// LS Electric XG5000 project: 4층_GEMINI
// PLC LSPLC
// module base 0 slot 0: 입출력 모듈:XBC-DR32H (DC 24V 입력, 릴레이 출력 32점)

PROGRAM 6 (task: 스캔 프로그램)

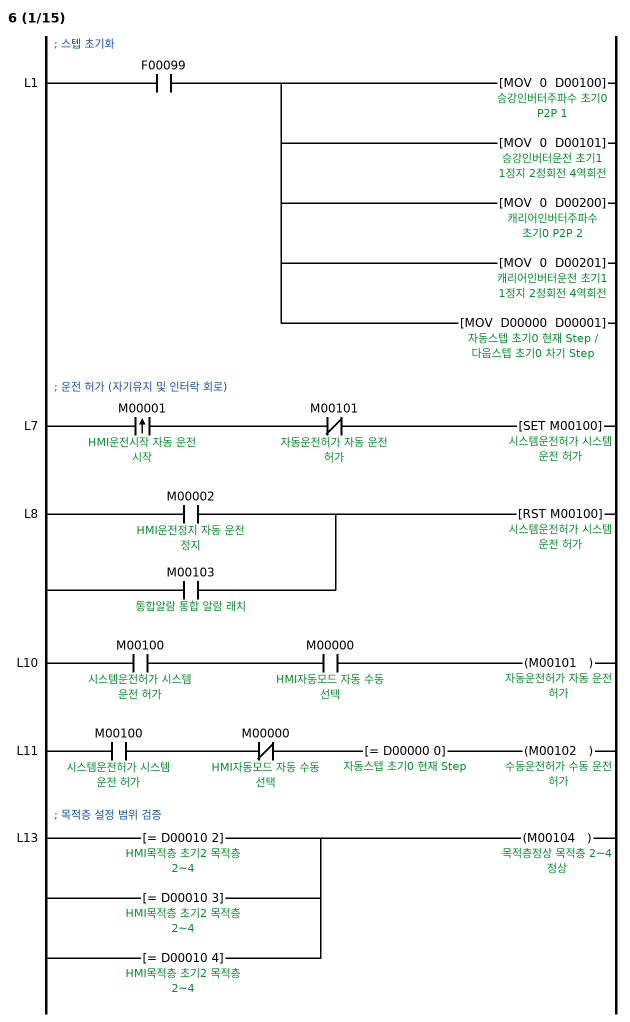
// 스텝 초기화
; L1
LOAD      F00099
MOV       0 D00100	// 승강인버터주파수 초기0 P2P 1
MOV       0 D00101	// 승강인버터운전 초기1 1정지 2정회전 4역회전
MOV       0 D00200	// 캐리어인버터주파수 초기0 P2P 2
MOV       0 D00201	// 캐리어인버터운전 초기1 1정지 2정회전 4역회전
MOV       D00000 D00001	// 자동스텝 초기0 현재 Step / 다음스텝 초기0 차기 Step
// 운전 허가 (자기유지 및 인터락 회로)
; L7
LOADP     M00001	// HMI운전시작 자동 운전 시작
AND NOT   M00101	// 자동운전허가 자동 운전 허가
SET       M00100	// 시스템운전허가 시스템 운전 허가
; L8
LOAD      M00002	// HMI운전정지 자동 운전 정지
OR        M00103	// 통합알람 통합 알람 래치
RST       M00100	// 시스템운전허가 시스템 운전 허가
; L10
LOAD      M00100	// 시스템운전허가 시스템 운전 허가
AND       M00000	// HMI자동모드 자동 수동 선택
OUT       M00101	// 자동운전허가 자동 운전 허가
; L11
LOAD      M00100	// 시스템운전허가 시스템 운전 허가
AND NOT   M00000	// HMI자동모드 자동 수동 선택
AND=      D00000 0	// 자동스텝 초기0 현재 Step
OUT       M00102	// 수동운전허가 수동 운전 허가
// 목적층 설정 범위 검증
; L13
LOAD=     D00010 2	// HMI목적층 초기2 목적층 2~4
OR=       D00010 3	// HMI목적층 초기2 목적층 2~4
OR=       D00010 4	// HMI목적층 초기2 목적층 2~4
OUT       M00104	// 목적층정상 목적층 2~4 정상

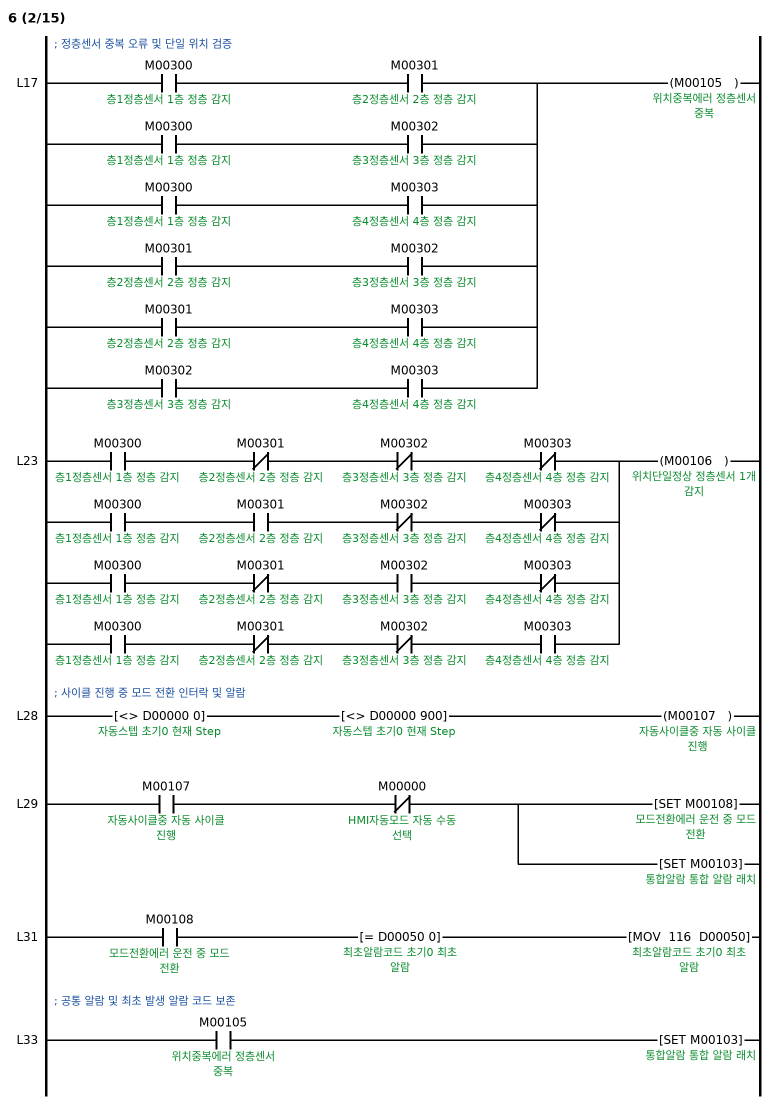
// 정층센서 중복 오류 및 단일 위치 검증
; L17
LOAD      M00300	// 층1정층센서 1층 정층 감지
AND       M00301	// 층2정층센서 2층 정층 감지
LOAD      M00300	// 층1정층센서 1층 정층 감지
AND       M00302	// 층3정층센서 3층 정층 감지
OR LOAD
LOAD      M00300	// 층1정층센서 1층 정층 감지
AND       M00303	// 층4정층센서 4층 정층 감지
OR LOAD
LOAD      M00301	// 층2정층센서 2층 정층 감지
AND       M00302	// 층3정층센서 3층 정층 감지
OR LOAD
LOAD      M00301	// 층2정층센서 2층 정층 감지
AND       M00303	// 층4정층센서 4층 정층 감지
OR LOAD
LOAD      M00302	// 층3정층센서 3층 정층 감지
AND       M00303	// 층4정층센서 4층 정층 감지
OR LOAD
OUT       M00105	// 위치중복에러 정층센서 중복
; L23
LOAD      M00300	// 층1정층센서 1층 정층 감지
AND NOT   M00301	// 층2정층센서 2층 정층 감지
AND NOT   M00302	// 층3정층센서 3층 정층 감지
AND NOT   M00303	// 층4정층센서 4층 정층 감지
LOAD      M00300	// 층1정층센서 1층 정층 감지
AND       M00301	// 층2정층센서 2층 정층 감지
AND NOT   M00302	// 층3정층센서 3층 정층 감지
AND NOT   M00303	// 층4정층센서 4층 정층 감지
OR LOAD
LOAD      M00300	// 층1정층센서 1층 정층 감지
AND NOT   M00301	// 층2정층센서 2층 정층 감지
AND       M00302	// 층3정층센서 3층 정층 감지
AND NOT   M00303	// 층4정층센서 4층 정층 감지
OR LOAD
LOAD      M00300	// 층1정층센서 1층 정층 감지
AND NOT   M00301	// 층2정층센서 2층 정층 감지
AND NOT   M00302	// 층3정층센서 3층 정층 감지
AND       M00303	// 층4정층센서 4층 정층 감지
OR LOAD
OUT       M00106	// 위치단일정상 정층센서 1개 감지
// 사이클 진행 중 모드 전환 인터락 및 알람
; L28
LOAD<>    D00000 0	// 자동스텝 초기0 현재 Step
AND<>     D00000 900	// 자동스텝 초기0 현재 Step
OUT       M00107	// 자동사이클중 자동 사이클 진행
; L29
LOAD      M00107	// 자동사이클중 자동 사이클 진행
AND NOT   M00000	// HMI자동모드 자동 수동 선택
SET       M00108	// 모드전환에러 운전 중 모드 전환
SET       M00103	// 통합알람 통합 알람 래치
; L31
LOAD      M00108	// 모드전환에러 운전 중 모드 전환
AND=      D00050 0	// 최초알람코드 초기0 최초 알람
MOV       116 D00050	// 최초알람코드 초기0 최초 알람
// 공통 알람 및 최초 발생 알람 코드 보존
; L33
LOAD      M00105	// 위치중복에러 정층센서 중복
SET       M00103	// 통합알람 통합 알람 래치

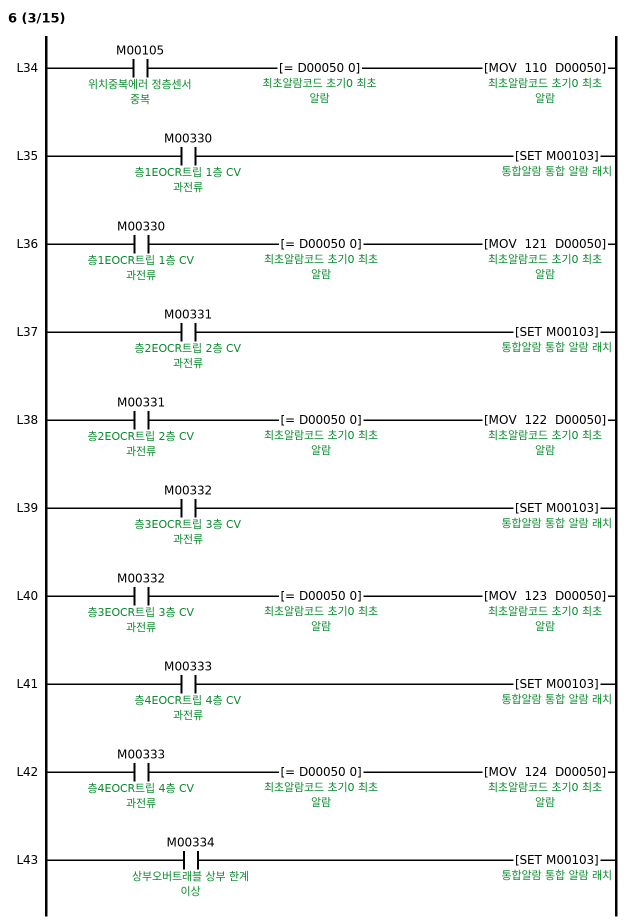
; L34
LOAD      M00105	// 위치중복에러 정층센서 중복
AND=      D00050 0	// 최초알람코드 초기0 최초 알람
MOV       110 D00050	// 최초알람코드 초기0 최초 알람
; L35
LOAD      M00330	// 층1EOCR트립 1층 CV 과전류
SET       M00103	// 통합알람 통합 알람 래치
; L36
LOAD      M00330	// 층1EOCR트립 1층 CV 과전류
AND=      D00050 0	// 최초알람코드 초기0 최초 알람
MOV       121 D00050	// 최초알람코드 초기0 최초 알람
; L37
LOAD      M00331	// 층2EOCR트립 2층 CV 과전류
SET       M00103	// 통합알람 통합 알람 래치
; L38
LOAD      M00331	// 층2EOCR트립 2층 CV 과전류
AND=      D00050 0	// 최초알람코드 초기0 최초 알람
MOV       122 D00050	// 최초알람코드 초기0 최초 알람
; L39
LOAD      M00332	// 층3EOCR트립 3층 CV 과전류
SET       M00103	// 통합알람 통합 알람 래치
; L40
LOAD      M00332	// 층3EOCR트립 3층 CV 과전류
AND=      D00050 0	// 최초알람코드 초기0 최초 알람
MOV       123 D00050	// 최초알람코드 초기0 최초 알람
; L41
LOAD      M00333	// 층4EOCR트립 4층 CV 과전류
SET       M00103	// 통합알람 통합 알람 래치
; L42
LOAD      M00333	// 층4EOCR트립 4층 CV 과전류
AND=      D00050 0	// 최초알람코드 초기0 최초 알람
MOV       124 D00050	// 최초알람코드 초기0 최초 알람
; L43
LOAD      M00334	// 상부오버트래블 상부 한계 이상
SET       M00103	// 통합알람 통합 알람 래치

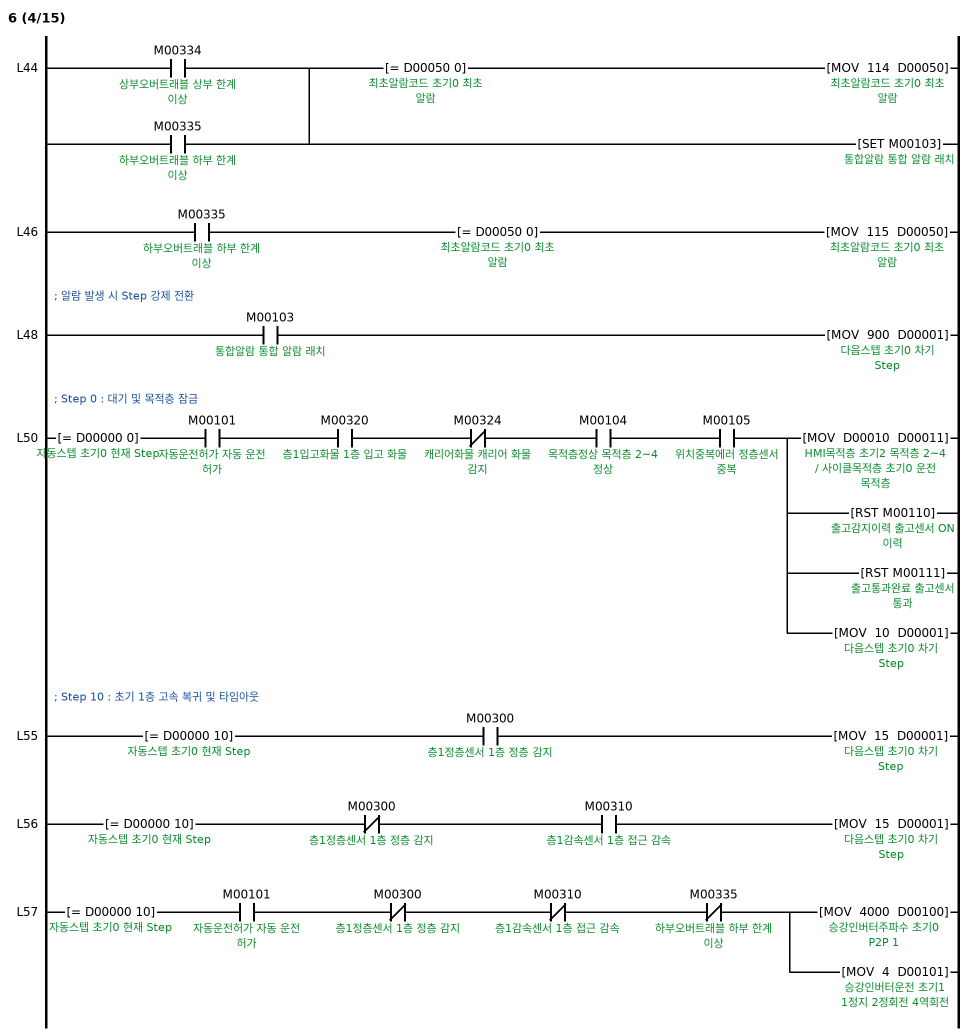
; L44
LOAD      M00334	// 상부오버트래블 상부 한계 이상
OR        M00335	// 하부오버트래블 하부 한계 이상
MPUSH
AND=      D00050 0	// 최초알람코드 초기0 최초 알람
MOV       114 D00050	// 최초알람코드 초기0 최초 알람
MPOP
SET       M00103	// 통합알람 통합 알람 래치
; L46
LOAD      M00335	// 하부오버트래블 하부 한계 이상
AND=      D00050 0	// 최초알람코드 초기0 최초 알람
MOV       115 D00050	// 최초알람코드 초기0 최초 알람
// 알람 발생 시 Step 강제 전환
; L48
LOAD      M00103	// 통합알람 통합 알람 래치
MOV       900 D00001	// 다음스텝 초기0 차기 Step
// Step 0 : 대기 및 목적층 잠금
; L50
LOAD=     D00000 0	// 자동스텝 초기0 현재 Step
AND       M00101	// 자동운전허가 자동 운전 허가
AND       M00320	// 층1입고화물 1층 입고 화물
AND NOT   M00324	// 캐리어화물 캐리어 화물 감지
AND       M00104	// 목적층정상 목적층 2~4 정상
AND       M00105	// 위치중복에러 정층센서 중복
MOV       D00010 D00011	// HMI목적층 초기2 목적층 2~4 / 사이클목적층 초기0 운전 목적층
RST       M00110	// 출고감지이력 출고센서 ON 이력
RST       M00111	// 출고통과완료 출고센서 통과
MOV       10 D00001	// 다음스텝 초기0 차기 Step
// Step 10 : 초기 1층 고속 복귀 및 타임아웃
; L55
LOAD=     D00000 10	// 자동스텝 초기0 현재 Step
AND       M00300	// 층1정층센서 1층 정층 감지
MOV       15 D00001	// 다음스텝 초기0 차기 Step
; L56
LOAD=     D00000 10	// 자동스텝 초기0 현재 Step
AND NOT   M00300	// 층1정층센서 1층 정층 감지
AND       M00310	// 층1감속센서 1층 접근 감속
MOV       15 D00001	// 다음스텝 초기0 차기 Step
; L57
LOAD=     D00000 10	// 자동스텝 초기0 현재 Step
AND       M00101	// 자동운전허가 자동 운전 허가
AND NOT   M00300	// 층1정층센서 1층 정층 감지
AND NOT   M00310	// 층1감속센서 1층 접근 감속
AND NOT   M00335	// 하부오버트래블 하부 한계 이상
MOV       4000 D00100	// 승강인버터주파수 초기0 P2P 1
MOV       4 D00101	// 승강인버터운전 초기1 1정지 2정회전 4역회전

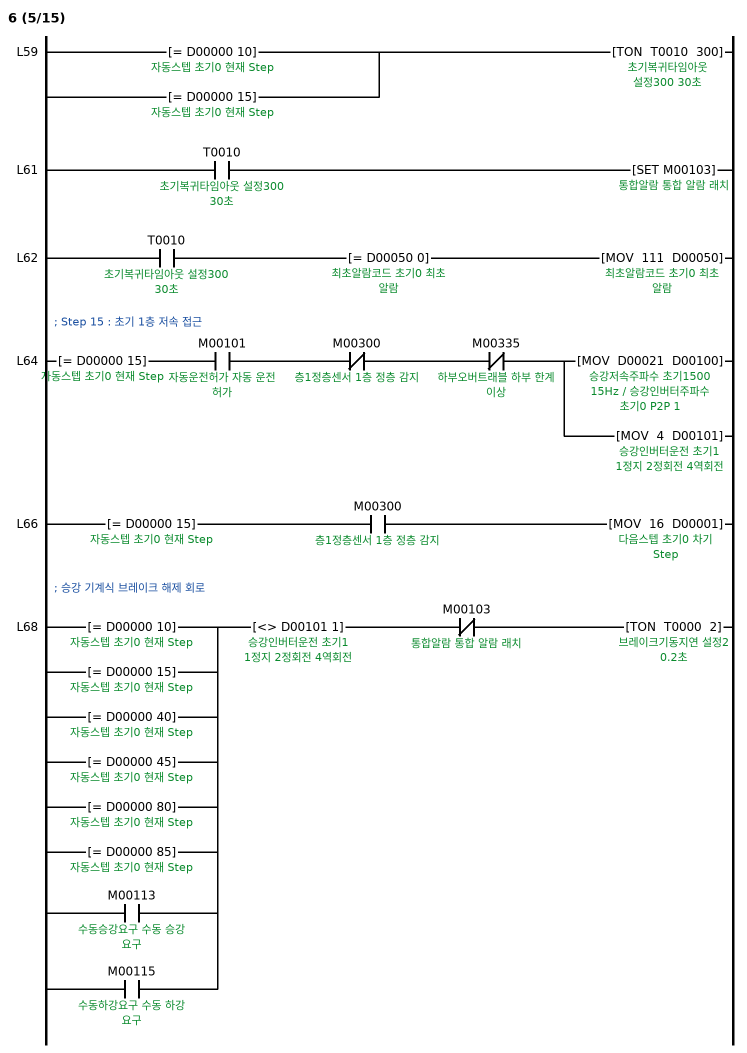
; L59
LOAD=     D00000 10	// 자동스텝 초기0 현재 Step
OR=       D00000 15	// 자동스텝 초기0 현재 Step
TON       T0010 300	// 초기복귀타임아웃 설정300 30초
; L61
LOAD      T0010	// 초기복귀타임아웃 설정300 30초
SET       M00103	// 통합알람 통합 알람 래치
; L62
LOAD      T0010	// 초기복귀타임아웃 설정300 30초
AND=      D00050 0	// 최초알람코드 초기0 최초 알람
MOV       111 D00050	// 최초알람코드 초기0 최초 알람
// Step 15 : 초기 1층 저속 접근
; L64
LOAD=     D00000 15	// 자동스텝 초기0 현재 Step
AND       M00101	// 자동운전허가 자동 운전 허가
AND NOT   M00300	// 층1정층센서 1층 정층 감지
AND NOT   M00335	// 하부오버트래블 하부 한계 이상
MOV       D00021 D00100	// 승강저속주파수 초기1500 15Hz / 승강인버터주파수 초기0 P2P 1
MOV       4 D00101	// 승강인버터운전 초기1 1정지 2정회전 4역회전
; L66
LOAD=     D00000 15	// 자동스텝 초기0 현재 Step
AND       M00300	// 층1정층센서 1층 정층 감지
MOV       16 D00001	// 다음스텝 초기0 차기 Step
// 승강 기계식 브레이크 해제 회로
; L68
LOAD=     D00000 10	// 자동스텝 초기0 현재 Step
OR=       D00000 15	// 자동스텝 초기0 현재 Step
OR=       D00000 40	// 자동스텝 초기0 현재 Step
OR=       D00000 45	// 자동스텝 초기0 현재 Step
OR=       D00000 80	// 자동스텝 초기0 현재 Step
OR=       D00000 85	// 자동스텝 초기0 현재 Step
OR        M00113	// 수동승강요구 수동 승강 요구
OR        M00115	// 수동하강요구 수동 하강 요구
AND<>     D00101 1	// 승강인버터운전 초기1 1정지 2정회전 4역회전
AND NOT   M00103	// 통합알람 통합 알람 래치
TON       T0000 2	// 브레이크기동지연 설정2 0.2초

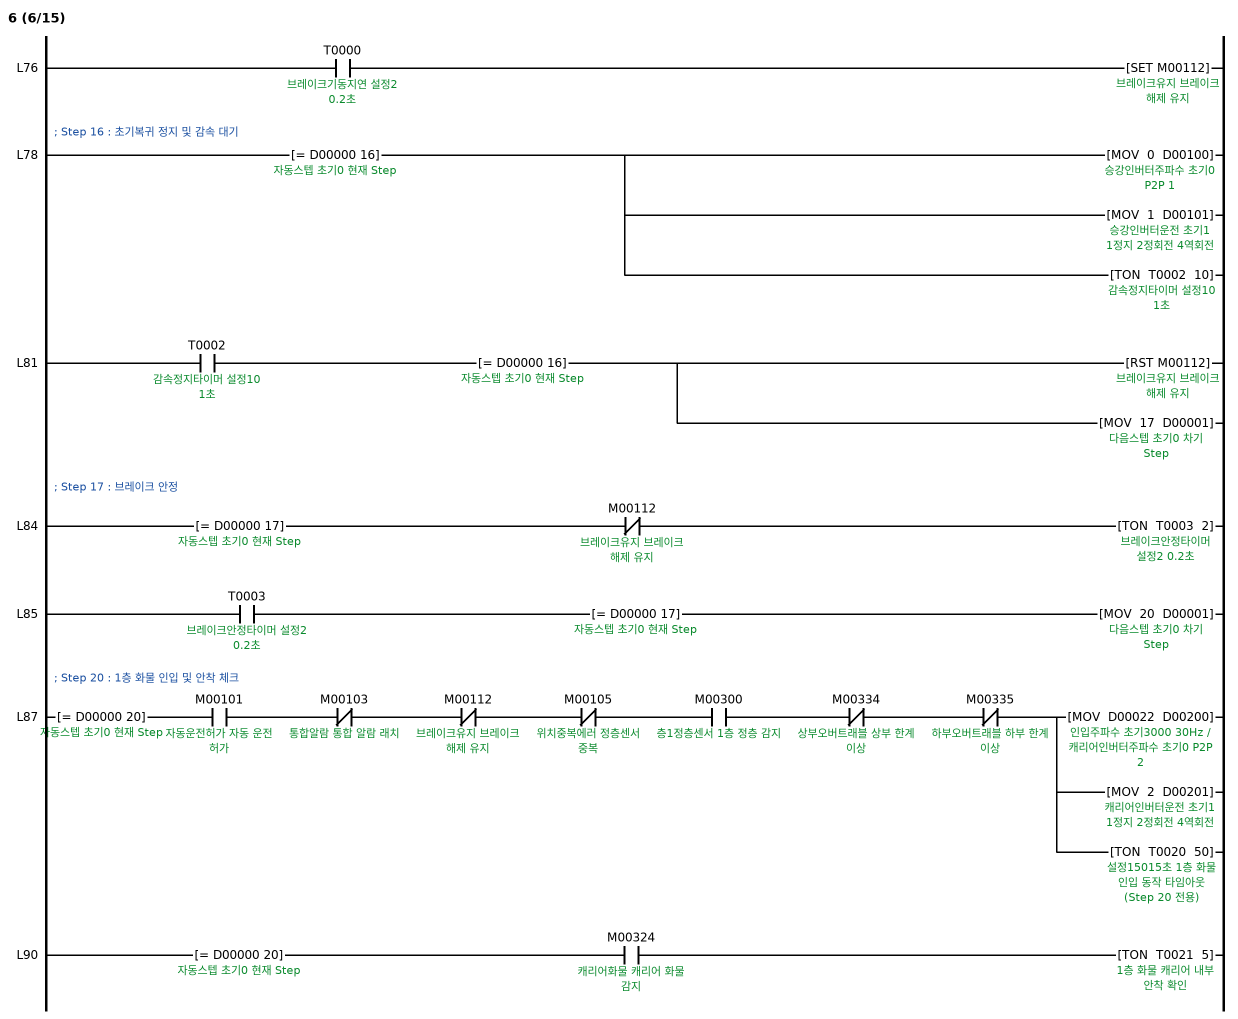
; L76
LOAD      T0000	// 브레이크기동지연 설정2 0.2초
SET       M00112	// 브레이크유지 브레이크 해제 유지
// Step 16 : 초기복귀 정지 및 감속 대기
; L78
LOAD=     D00000 16	// 자동스텝 초기0 현재 Step
MOV       0 D00100	// 승강인버터주파수 초기0 P2P 1
MOV       1 D00101	// 승강인버터운전 초기1 1정지 2정회전 4역회전
TON       T0002 10	// 감속정지타이머 설정10 1초
; L81
LOAD      T0002	// 감속정지타이머 설정10 1초
AND=      D00000 16	// 자동스텝 초기0 현재 Step
RST       M00112	// 브레이크유지 브레이크 해제 유지
MOV       17 D00001	// 다음스텝 초기0 차기 Step
// Step 17 : 브레이크 안정
; L84
LOAD=     D00000 17	// 자동스텝 초기0 현재 Step
AND NOT   M00112	// 브레이크유지 브레이크 해제 유지
TON       T0003 2	// 브레이크안정타이머 설정2 0.2초
; L85
LOAD      T0003	// 브레이크안정타이머 설정2 0.2초
AND=      D00000 17	// 자동스텝 초기0 현재 Step
MOV       20 D00001	// 다음스텝 초기0 차기 Step
// Step 20 : 1층 화물 인입 및 안착 체크
; L87
LOAD=     D00000 20	// 자동스텝 초기0 현재 Step
AND       M00101	// 자동운전허가 자동 운전 허가
AND NOT   M00103	// 통합알람 통합 알람 래치
AND NOT   M00112	// 브레이크유지 브레이크 해제 유지
AND NOT   M00105	// 위치중복에러 정층센서 중복
AND       M00300	// 층1정층센서 1층 정층 감지
AND NOT   M00334	// 상부오버트래블 상부 한계 이상
AND NOT   M00335	// 하부오버트래블 하부 한계 이상
MOV       D00022 D00200	// 인입주파수 초기3000 30Hz / 캐리어인버터주파수 초기0 P2P 2
MOV       2 D00201	// 캐리어인버터운전 초기1 1정지 2정회전 4역회전
TON       T0020 50	// 설정15015초 1층 화물 인입 동작 타임아웃 (Step 20 전용)
; L90
LOAD=     D00000 20	// 자동스텝 초기0 현재 Step
AND       M00324	// 캐리어화물 캐리어 화물 감지
TON       T0021 5	// 1층 화물 캐리어 내부 안착 확인

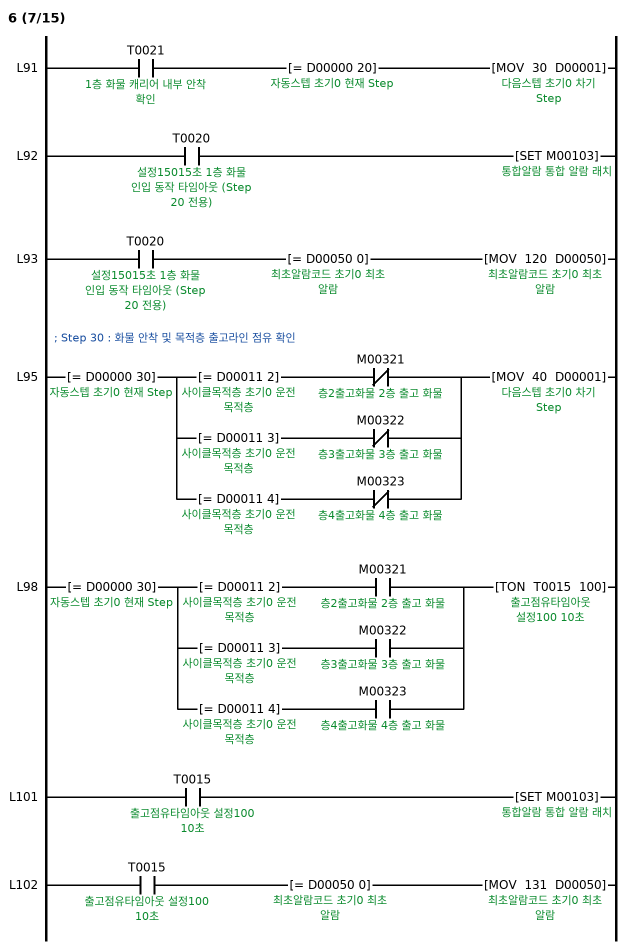
; L91
LOAD      T0021	// 1층 화물 캐리어 내부 안착 확인
AND=      D00000 20	// 자동스텝 초기0 현재 Step
MOV       30 D00001	// 다음스텝 초기0 차기 Step
; L92
LOAD      T0020	// 설정15015초 1층 화물 인입 동작 타임아웃 (Step 20 전용)
SET       M00103	// 통합알람 통합 알람 래치
; L93
LOAD      T0020	// 설정15015초 1층 화물 인입 동작 타임아웃 (Step 20 전용)
AND=      D00050 0	// 최초알람코드 초기0 최초 알람
MOV       120 D00050	// 최초알람코드 초기0 최초 알람
// Step 30 : 화물 안착 및 목적층 출고라인 점유 확인
; L95
LOAD=     D00000 30	// 자동스텝 초기0 현재 Step
LOAD=     D00011 2	// 사이클목적층 초기0 운전 목적층
AND NOT   M00321	// 층2출고화물 2층 출고 화물
LOAD=     D00011 3	// 사이클목적층 초기0 운전 목적층
AND NOT   M00322	// 층3출고화물 3층 출고 화물
OR LOAD
LOAD=     D00011 4	// 사이클목적층 초기0 운전 목적층
AND NOT   M00323	// 층4출고화물 4층 출고 화물
OR LOAD
AND LOAD
MOV       40 D00001	// 다음스텝 초기0 차기 Step
; L98
LOAD=     D00000 30	// 자동스텝 초기0 현재 Step
LOAD=     D00011 2	// 사이클목적층 초기0 운전 목적층
AND       M00321	// 층2출고화물 2층 출고 화물
LOAD=     D00011 3	// 사이클목적층 초기0 운전 목적층
AND       M00322	// 층3출고화물 3층 출고 화물
OR LOAD
LOAD=     D00011 4	// 사이클목적층 초기0 운전 목적층
AND       M00323	// 층4출고화물 4층 출고 화물
OR LOAD
AND LOAD
TON       T0015 100	// 출고점유타임아웃 설정100 10초
; L101
LOAD      T0015	// 출고점유타임아웃 설정100 10초
SET       M00103	// 통합알람 통합 알람 래치
; L102
LOAD      T0015	// 출고점유타임아웃 설정100 10초
AND=      D00050 0	// 최초알람코드 초기0 최초 알람
MOV       131 D00050	// 최초알람코드 초기0 최초 알람

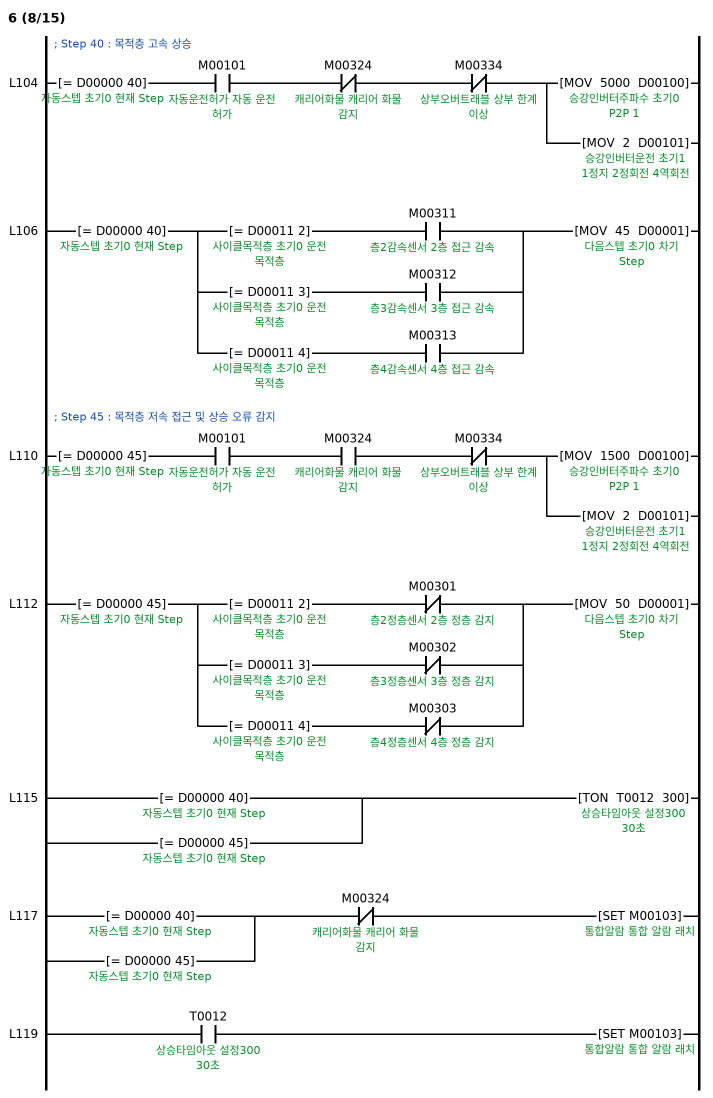
// Step 40 : 목적층 고속 상승
; L104
LOAD=     D00000 40	// 자동스텝 초기0 현재 Step
AND       M00101	// 자동운전허가 자동 운전 허가
AND NOT   M00324	// 캐리어화물 캐리어 화물 감지
AND NOT   M00334	// 상부오버트래블 상부 한계 이상
MOV       5000 D00100	// 승강인버터주파수 초기0 P2P 1
MOV       2 D00101	// 승강인버터운전 초기1 1정지 2정회전 4역회전
; L106
LOAD=     D00000 40	// 자동스텝 초기0 현재 Step
LOAD=     D00011 2	// 사이클목적층 초기0 운전 목적층
AND       M00311	// 층2감속센서 2층 접근 감속
LOAD=     D00011 3	// 사이클목적층 초기0 운전 목적층
AND       M00312	// 층3감속센서 3층 접근 감속
OR LOAD
LOAD=     D00011 4	// 사이클목적층 초기0 운전 목적층
AND       M00313	// 층4감속센서 4층 접근 감속
OR LOAD
AND LOAD
MOV       45 D00001	// 다음스텝 초기0 차기 Step
// Step 45 : 목적층 저속 접근 및 상승 오류 감지
; L110
LOAD=     D00000 45	// 자동스텝 초기0 현재 Step
AND       M00101	// 자동운전허가 자동 운전 허가
AND       M00324	// 캐리어화물 캐리어 화물 감지
AND NOT   M00334	// 상부오버트래블 상부 한계 이상
MOV       1500 D00100	// 승강인버터주파수 초기0 P2P 1
MOV       2 D00101	// 승강인버터운전 초기1 1정지 2정회전 4역회전
; L112
LOAD=     D00000 45	// 자동스텝 초기0 현재 Step
LOAD=     D00011 2	// 사이클목적층 초기0 운전 목적층
AND NOT   M00301	// 층2정층센서 2층 정층 감지
LOAD=     D00011 3	// 사이클목적층 초기0 운전 목적층
AND NOT   M00302	// 층3정층센서 3층 정층 감지
OR LOAD
LOAD=     D00011 4	// 사이클목적층 초기0 운전 목적층
AND NOT   M00303	// 층4정층센서 4층 정층 감지
OR LOAD
AND LOAD
MOV       50 D00001	// 다음스텝 초기0 차기 Step
; L115
LOAD=     D00000 40	// 자동스텝 초기0 현재 Step
OR=       D00000 45	// 자동스텝 초기0 현재 Step
TON       T0012 300	// 상승타임아웃 설정300 30초
; L117
LOAD=     D00000 40	// 자동스텝 초기0 현재 Step
OR=       D00000 45	// 자동스텝 초기0 현재 Step
AND NOT   M00324	// 캐리어화물 캐리어 화물 감지
SET       M00103	// 통합알람 통합 알람 래치
; L119
LOAD      T0012	// 상승타임아웃 설정300 30초
SET       M00103	// 통합알람 통합 알람 래치

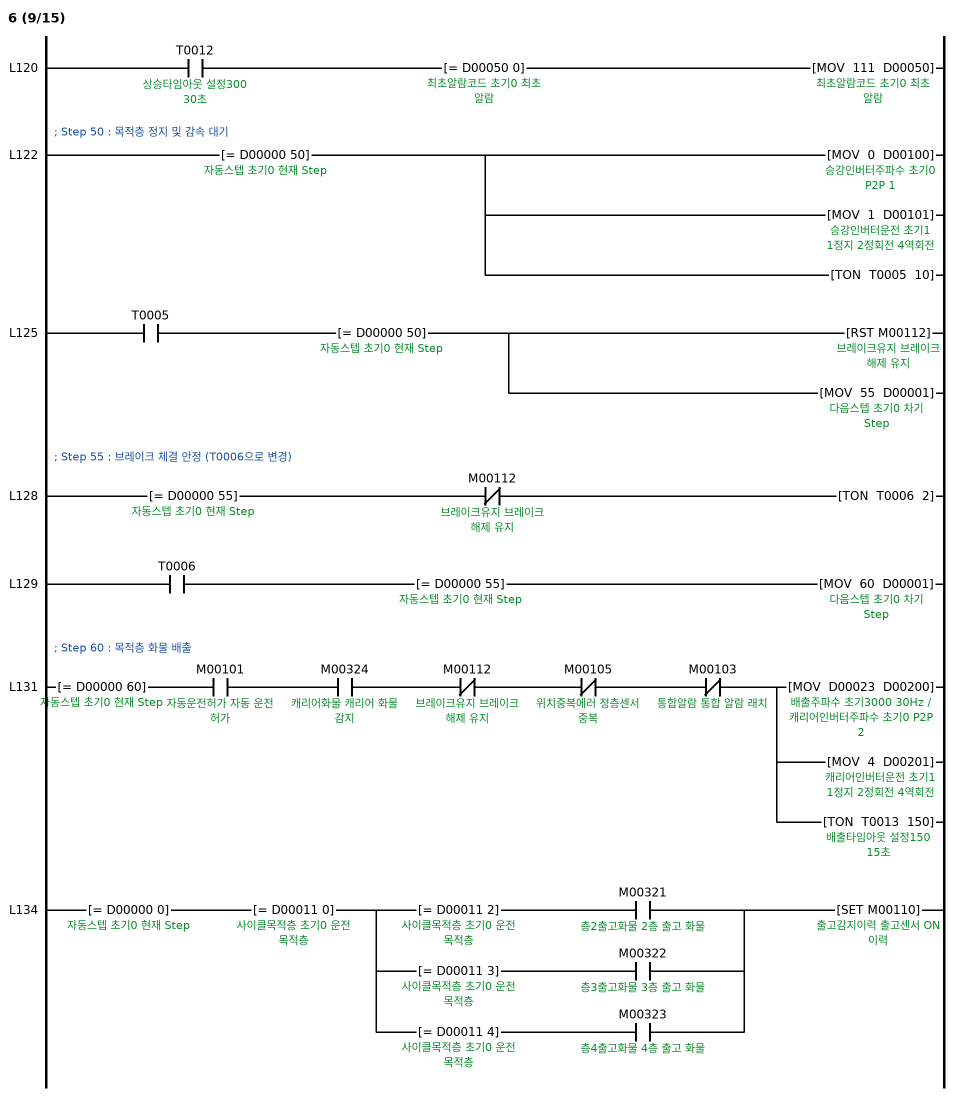
; L120
LOAD      T0012	// 상승타임아웃 설정300 30초
AND=      D00050 0	// 최초알람코드 초기0 최초 알람
MOV       111 D00050	// 최초알람코드 초기0 최초 알람
// Step 50 : 목적층 정지 및 감속 대기
; L122
LOAD=     D00000 50	// 자동스텝 초기0 현재 Step
MOV       0 D00100	// 승강인버터주파수 초기0 P2P 1
MOV       1 D00101	// 승강인버터운전 초기1 1정지 2정회전 4역회전
TON       T0005 10
; L125
LOAD      T0005
AND=      D00000 50	// 자동스텝 초기0 현재 Step
RST       M00112	// 브레이크유지 브레이크 해제 유지
MOV       55 D00001	// 다음스텝 초기0 차기 Step
// Step 55 : 브레이크 체결 안정 (T0006으로 변경)
; L128
LOAD=     D00000 55	// 자동스텝 초기0 현재 Step
AND NOT   M00112	// 브레이크유지 브레이크 해제 유지
TON       T0006 2
; L129
LOAD      T0006
AND=      D00000 55	// 자동스텝 초기0 현재 Step
MOV       60 D00001	// 다음스텝 초기0 차기 Step
// Step 60 : 목적층 화물 배출
; L131
LOAD=     D00000 60	// 자동스텝 초기0 현재 Step
AND       M00101	// 자동운전허가 자동 운전 허가
AND       M00324	// 캐리어화물 캐리어 화물 감지
AND NOT   M00112	// 브레이크유지 브레이크 해제 유지
AND NOT   M00105	// 위치중복에러 정층센서 중복
AND NOT   M00103	// 통합알람 통합 알람 래치
MOV       D00023 D00200	// 배출주파수 초기3000 30Hz / 캐리어인버터주파수 초기0 P2P 2
MOV       4 D00201	// 캐리어인버터운전 초기1 1정지 2정회전 4역회전
TON       T0013 150	// 배출타임아웃 설정150 15초
; L134
LOAD=     D00000 0	// 자동스텝 초기0 현재 Step
AND=      D00011 0	// 사이클목적층 초기0 운전 목적층
LOAD=     D00011 2	// 사이클목적층 초기0 운전 목적층
AND       M00321	// 층2출고화물 2층 출고 화물
LOAD=     D00011 3	// 사이클목적층 초기0 운전 목적층
AND       M00322	// 층3출고화물 3층 출고 화물
OR LOAD
LOAD=     D00011 4	// 사이클목적층 초기0 운전 목적층
AND       M00323	// 층4출고화물 4층 출고 화물
OR LOAD
AND LOAD
SET       M00110	// 출고감지이력 출고센서 ON 이력

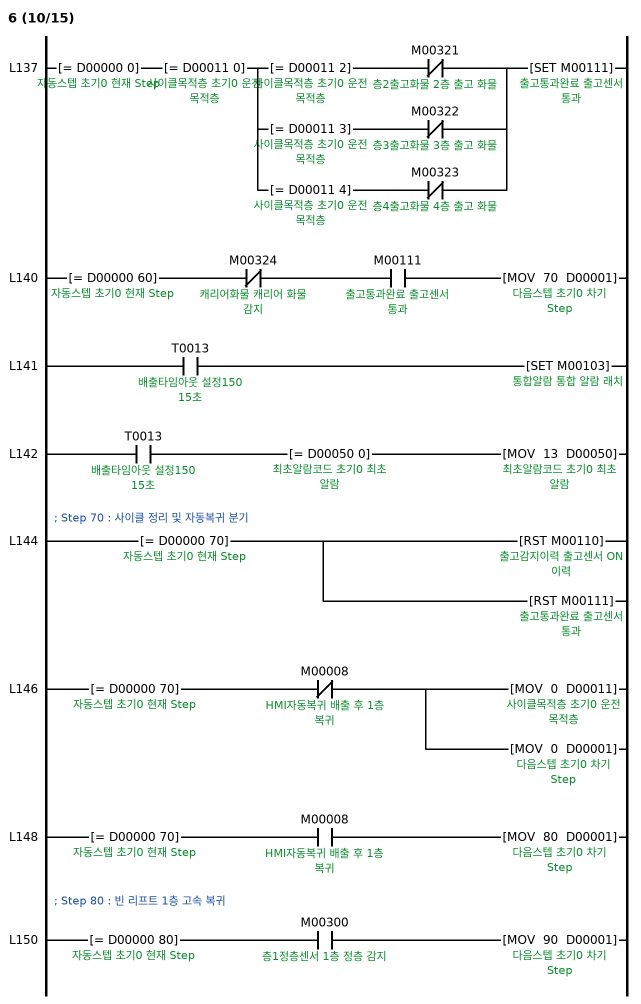
; L137
LOAD=     D00000 0	// 자동스텝 초기0 현재 Step
AND=      D00011 0	// 사이클목적층 초기0 운전 목적층
LOAD=     D00011 2	// 사이클목적층 초기0 운전 목적층
AND NOT   M00321	// 층2출고화물 2층 출고 화물
LOAD=     D00011 3	// 사이클목적층 초기0 운전 목적층
AND NOT   M00322	// 층3출고화물 3층 출고 화물
OR LOAD
LOAD=     D00011 4	// 사이클목적층 초기0 운전 목적층
AND NOT   M00323	// 층4출고화물 4층 출고 화물
OR LOAD
AND LOAD
SET       M00111	// 출고통과완료 출고센서 통과
; L140
LOAD=     D00000 60	// 자동스텝 초기0 현재 Step
AND NOT   M00324	// 캐리어화물 캐리어 화물 감지
AND       M00111	// 출고통과완료 출고센서 통과
MOV       70 D00001	// 다음스텝 초기0 차기 Step
; L141
LOAD      T0013	// 배출타임아웃 설정150 15초
SET       M00103	// 통합알람 통합 알람 래치
; L142
LOAD      T0013	// 배출타임아웃 설정150 15초
AND=      D00050 0	// 최초알람코드 초기0 최초 알람
MOV       13 D00050	// 최초알람코드 초기0 최초 알람
// Step 70 : 사이클 정리 및 자동복귀 분기
; L144
LOAD=     D00000 70	// 자동스텝 초기0 현재 Step
RST       M00110	// 출고감지이력 출고센서 ON 이력
RST       M00111	// 출고통과완료 출고센서 통과
; L146
LOAD=     D00000 70	// 자동스텝 초기0 현재 Step
AND NOT   M00008	// HMI자동복귀 배출 후 1층 복귀
MOV       0 D00011	// 사이클목적층 초기0 운전 목적층
MOV       0 D00001	// 다음스텝 초기0 차기 Step
; L148
LOAD=     D00000 70	// 자동스텝 초기0 현재 Step
AND       M00008	// HMI자동복귀 배출 후 1층 복귀
MOV       80 D00001	// 다음스텝 초기0 차기 Step
// Step 80 : 빈 리프트 1층 고속 복귀
; L150
LOAD=     D00000 80	// 자동스텝 초기0 현재 Step
AND       M00300	// 층1정층센서 1층 정층 감지
MOV       90 D00001	// 다음스텝 초기0 차기 Step

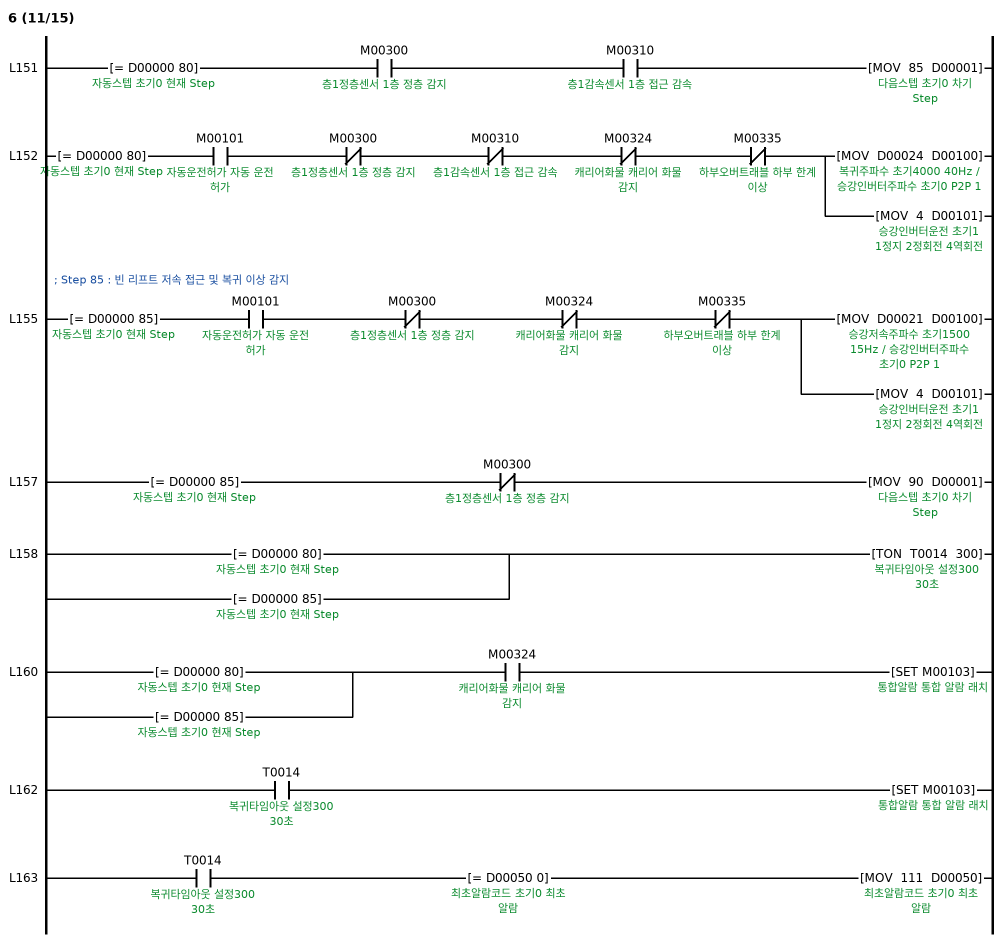
; L151
LOAD=     D00000 80	// 자동스텝 초기0 현재 Step
AND       M00300	// 층1정층센서 1층 정층 감지
AND       M00310	// 층1감속센서 1층 접근 감속
MOV       85 D00001	// 다음스텝 초기0 차기 Step
; L152
LOAD=     D00000 80	// 자동스텝 초기0 현재 Step
AND       M00101	// 자동운전허가 자동 운전 허가
AND NOT   M00300	// 층1정층센서 1층 정층 감지
AND NOT   M00310	// 층1감속센서 1층 접근 감속
AND NOT   M00324	// 캐리어화물 캐리어 화물 감지
AND NOT   M00335	// 하부오버트래블 하부 한계 이상
MOV       D00024 D00100	// 복귀주파수 초기4000 40Hz / 승강인버터주파수 초기0 P2P 1
MOV       4 D00101	// 승강인버터운전 초기1 1정지 2정회전 4역회전
// Step 85 : 빈 리프트 저속 접근 및 복귀 이상 감지
; L155
LOAD=     D00000 85	// 자동스텝 초기0 현재 Step
AND       M00101	// 자동운전허가 자동 운전 허가
AND NOT   M00300	// 층1정층센서 1층 정층 감지
AND NOT   M00324	// 캐리어화물 캐리어 화물 감지
AND NOT   M00335	// 하부오버트래블 하부 한계 이상
MOV       D00021 D00100	// 승강저속주파수 초기1500 15Hz / 승강인버터주파수 초기0 P2P 1
MOV       4 D00101	// 승강인버터운전 초기1 1정지 2정회전 4역회전
; L157
LOAD=     D00000 85	// 자동스텝 초기0 현재 Step
AND NOT   M00300	// 층1정층센서 1층 정층 감지
MOV       90 D00001	// 다음스텝 초기0 차기 Step
; L158
LOAD=     D00000 80	// 자동스텝 초기0 현재 Step
OR=       D00000 85	// 자동스텝 초기0 현재 Step
TON       T0014 300	// 복귀타임아웃 설정300 30초
; L160
LOAD=     D00000 80	// 자동스텝 초기0 현재 Step
OR=       D00000 85	// 자동스텝 초기0 현재 Step
AND       M00324	// 캐리어화물 캐리어 화물 감지
SET       M00103	// 통합알람 통합 알람 래치
; L162
LOAD      T0014	// 복귀타임아웃 설정300 30초
SET       M00103	// 통합알람 통합 알람 래치
; L163
LOAD      T0014	// 복귀타임아웃 설정300 30초
AND=      D00050 0	// 최초알람코드 초기0 최초 알람
MOV       111 D00050	// 최초알람코드 초기0 최초 알람

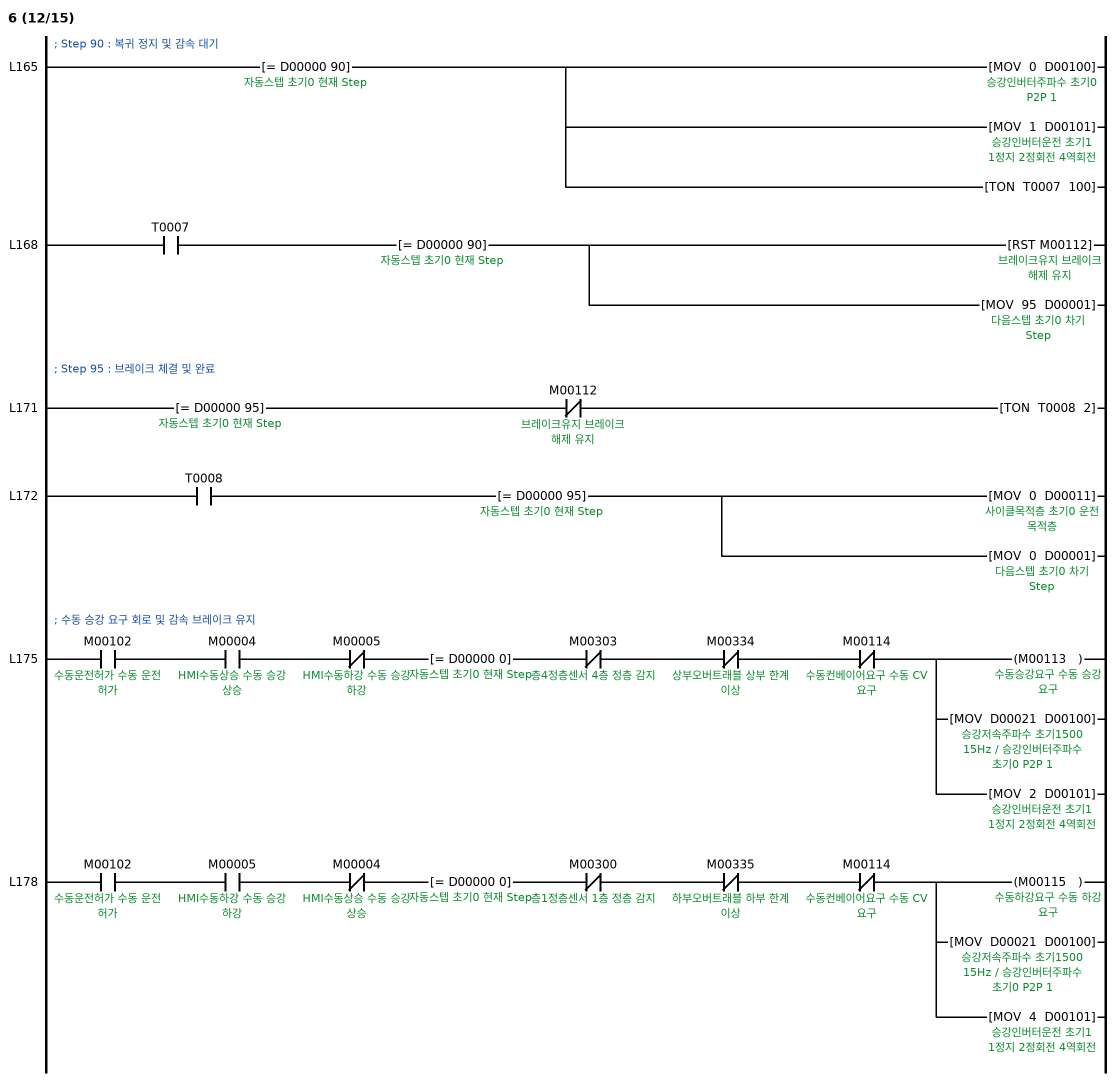
// Step 90 : 복귀 정지 및 감속 대기
; L165
LOAD=     D00000 90	// 자동스텝 초기0 현재 Step
MOV       0 D00100	// 승강인버터주파수 초기0 P2P 1
MOV       1 D00101	// 승강인버터운전 초기1 1정지 2정회전 4역회전
TON       T0007 100
; L168
LOAD      T0007
AND=      D00000 90	// 자동스텝 초기0 현재 Step
RST       M00112	// 브레이크유지 브레이크 해제 유지
MOV       95 D00001	// 다음스텝 초기0 차기 Step
// Step 95 : 브레이크 체결 및 완료
; L171
LOAD=     D00000 95	// 자동스텝 초기0 현재 Step
AND NOT   M00112	// 브레이크유지 브레이크 해제 유지
TON       T0008 2
; L172
LOAD      T0008
AND=      D00000 95	// 자동스텝 초기0 현재 Step
MOV       0 D00011	// 사이클목적층 초기0 운전 목적층
MOV       0 D00001	// 다음스텝 초기0 차기 Step
// 수동 승강 요구 회로 및 감속 브레이크 유지
; L175
LOAD      M00102	// 수동운전허가 수동 운전 허가
AND       M00004	// HMI수동상승 수동 승강 상승
AND NOT   M00005	// HMI수동하강 수동 승강 하강
AND=      D00000 0	// 자동스텝 초기0 현재 Step
AND NOT   M00303	// 층4정층센서 4층 정층 감지
AND NOT   M00334	// 상부오버트래블 상부 한계 이상
AND NOT   M00114	// 수동컨베이어요구 수동 CV 요구
OUT       M00113	// 수동승강요구 수동 승강 요구
MOV       D00021 D00100	// 승강저속주파수 초기1500 15Hz / 승강인버터주파수 초기0 P2P 1
MOV       2 D00101	// 승강인버터운전 초기1 1정지 2정회전 4역회전
; L178
LOAD      M00102	// 수동운전허가 수동 운전 허가
AND       M00005	// HMI수동하강 수동 승강 하강
AND NOT   M00004	// HMI수동상승 수동 승강 상승
AND=      D00000 0	// 자동스텝 초기0 현재 Step
AND NOT   M00300	// 층1정층센서 1층 정층 감지
AND NOT   M00335	// 하부오버트래블 하부 한계 이상
AND NOT   M00114	// 수동컨베이어요구 수동 CV 요구
OUT       M00115	// 수동하강요구 수동 하강 요구
MOV       D00021 D00100	// 승강저속주파수 초기1500 15Hz / 승강인버터주파수 초기0 P2P 1
MOV       4 D00101	// 승강인버터운전 초기1 1정지 2정회전 4역회전

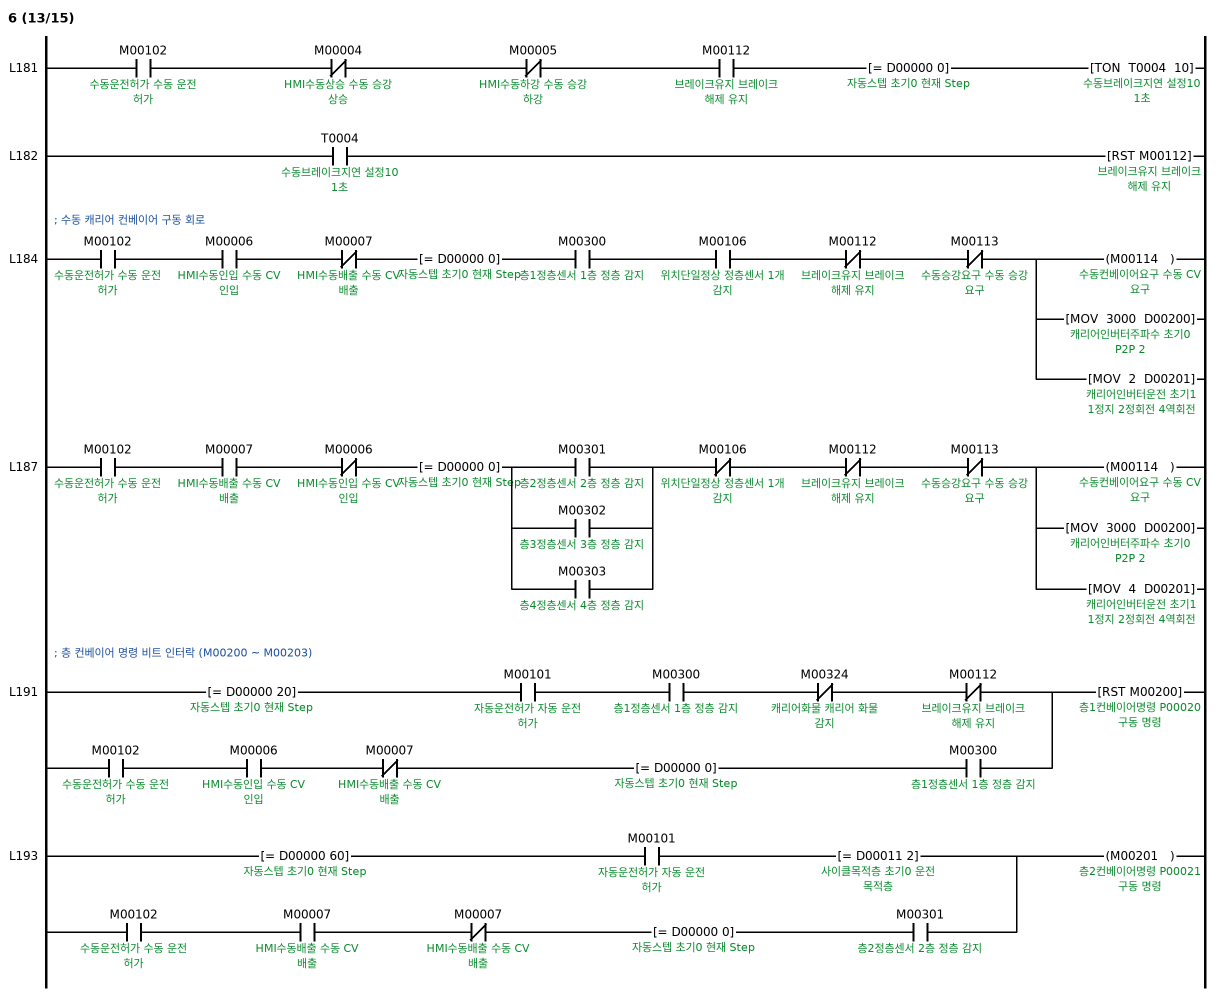
; L181
LOAD      M00102	// 수동운전허가 수동 운전 허가
AND NOT   M00004	// HMI수동상승 수동 승강 상승
AND NOT   M00005	// HMI수동하강 수동 승강 하강
AND       M00112	// 브레이크유지 브레이크 해제 유지
AND=      D00000 0	// 자동스텝 초기0 현재 Step
TON       T0004 10	// 수동브레이크지연 설정10 1초
; L182
LOAD      T0004	// 수동브레이크지연 설정10 1초
RST       M00112	// 브레이크유지 브레이크 해제 유지
// 수동 캐리어 컨베이어 구동 회로
; L184
LOAD      M00102	// 수동운전허가 수동 운전 허가
AND       M00006	// HMI수동인입 수동 CV 인입
AND NOT   M00007	// HMI수동배출 수동 CV 배출
AND=      D00000 0	// 자동스텝 초기0 현재 Step
AND       M00300	// 층1정층센서 1층 정층 감지
AND       M00106	// 위치단일정상 정층센서 1개 감지
AND NOT   M00112	// 브레이크유지 브레이크 해제 유지
AND NOT   M00113	// 수동승강요구 수동 승강 요구
OUT       M00114	// 수동컨베이어요구 수동 CV 요구
MOV       3000 D00200	// 캐리어인버터주파수 초기0 P2P 2
MOV       2 D00201	// 캐리어인버터운전 초기1 1정지 2정회전 4역회전
; L187
LOAD      M00102	// 수동운전허가 수동 운전 허가
AND       M00007	// HMI수동배출 수동 CV 배출
AND NOT   M00006	// HMI수동인입 수동 CV 인입
AND=      D00000 0	// 자동스텝 초기0 현재 Step
LOAD      M00301	// 층2정층센서 2층 정층 감지
OR        M00302	// 층3정층센서 3층 정층 감지
OR        M00303	// 층4정층센서 4층 정층 감지
AND LOAD
AND NOT   M00106	// 위치단일정상 정층센서 1개 감지
AND NOT   M00112	// 브레이크유지 브레이크 해제 유지
AND NOT   M00113	// 수동승강요구 수동 승강 요구
OUT       M00114	// 수동컨베이어요구 수동 CV 요구
MOV       3000 D00200	// 캐리어인버터주파수 초기0 P2P 2
MOV       4 D00201	// 캐리어인버터운전 초기1 1정지 2정회전 4역회전
// 층 컨베이어 명령 비트 인터락 (M00200 ~ M00203)
; L191
LOAD=     D00000 20	// 자동스텝 초기0 현재 Step
AND       M00101	// 자동운전허가 자동 운전 허가
AND       M00300	// 층1정층센서 1층 정층 감지
AND NOT   M00324	// 캐리어화물 캐리어 화물 감지
AND NOT   M00112	// 브레이크유지 브레이크 해제 유지
LOAD      M00102	// 수동운전허가 수동 운전 허가
AND       M00006	// HMI수동인입 수동 CV 인입
AND NOT   M00007	// HMI수동배출 수동 CV 배출
AND=      D00000 0	// 자동스텝 초기0 현재 Step
AND       M00300	// 층1정층센서 1층 정층 감지
OR LOAD
RST       M00200	// 층1컨베이어명령 P00020 구동 명령
; L193
LOAD=     D00000 60	// 자동스텝 초기0 현재 Step
AND       M00101	// 자동운전허가 자동 운전 허가
AND=      D00011 2	// 사이클목적층 초기0 운전 목적층
LOAD      M00102	// 수동운전허가 수동 운전 허가
AND       M00007	// HMI수동배출 수동 CV 배출
AND NOT   M00007	// HMI수동배출 수동 CV 배출
AND=      D00000 0	// 자동스텝 초기0 현재 Step
AND       M00301	// 층2정층센서 2층 정층 감지
OR LOAD
OUT       M00201	// 층2컨베이어명령 P00021 구동 명령

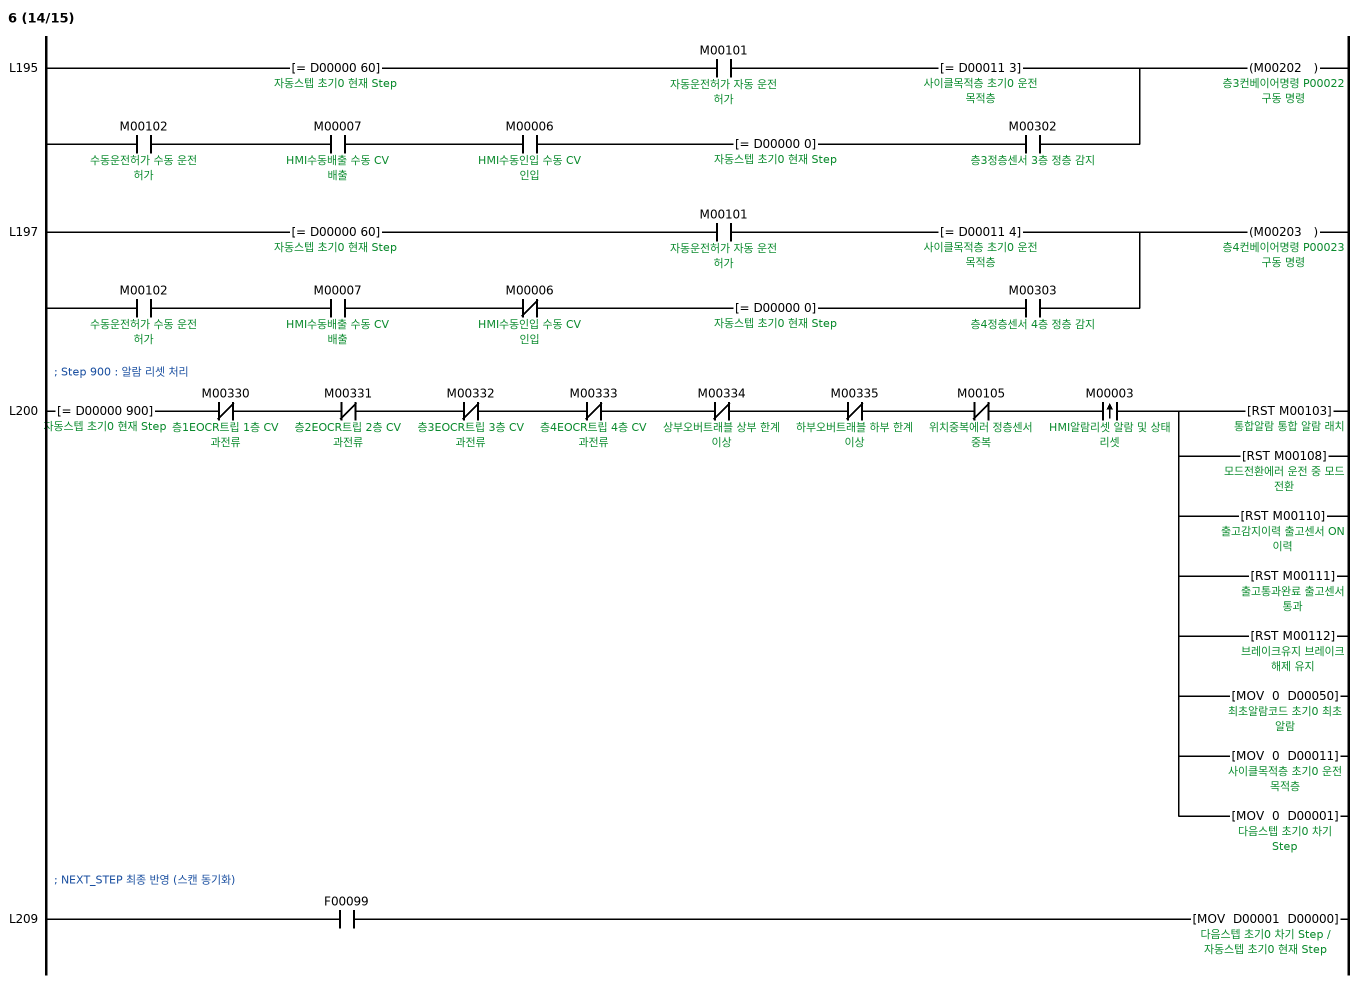
; L195
LOAD=     D00000 60	// 자동스텝 초기0 현재 Step
AND       M00101	// 자동운전허가 자동 운전 허가
AND=      D00011 3	// 사이클목적층 초기0 운전 목적층
LOAD      M00102	// 수동운전허가 수동 운전 허가
AND       M00007	// HMI수동배출 수동 CV 배출
AND       M00006	// HMI수동인입 수동 CV 인입
AND=      D00000 0	// 자동스텝 초기0 현재 Step
AND       M00302	// 층3정층센서 3층 정층 감지
OR LOAD
OUT       M00202	// 층3컨베이어명령 P00022 구동 명령
; L197
LOAD=     D00000 60	// 자동스텝 초기0 현재 Step
AND       M00101	// 자동운전허가 자동 운전 허가
AND=      D00011 4	// 사이클목적층 초기0 운전 목적층
LOAD      M00102	// 수동운전허가 수동 운전 허가
AND       M00007	// HMI수동배출 수동 CV 배출
AND NOT   M00006	// HMI수동인입 수동 CV 인입
AND=      D00000 0	// 자동스텝 초기0 현재 Step
AND       M00303	// 층4정층센서 4층 정층 감지
OR LOAD
OUT       M00203	// 층4컨베이어명령 P00023 구동 명령
// Step 900 : 알람 리셋 처리
; L200
LOAD=     D00000 900	// 자동스텝 초기0 현재 Step
AND NOT   M00330	// 층1EOCR트립 1층 CV 과전류
AND NOT   M00331	// 층2EOCR트립 2층 CV 과전류
AND NOT   M00332	// 층3EOCR트립 3층 CV 과전류
AND NOT   M00333	// 층4EOCR트립 4층 CV 과전류
AND NOT   M00334	// 상부오버트래블 상부 한계 이상
AND NOT   M00335	// 하부오버트래블 하부 한계 이상
AND NOT   M00105	// 위치중복에러 정층센서 중복
ANDP      M00003	// HMI알람리셋 알람 및 상태 리셋
RST       M00103	// 통합알람 통합 알람 래치
RST       M00108	// 모드전환에러 운전 중 모드 전환
RST       M00110	// 출고감지이력 출고센서 ON 이력
RST       M00111	// 출고통과완료 출고센서 통과
RST       M00112	// 브레이크유지 브레이크 해제 유지
MOV       0 D00050	// 최초알람코드 초기0 최초 알람
MOV       0 D00011	// 사이클목적층 초기0 운전 목적층
MOV       0 D00001	// 다음스텝 초기0 차기 Step
// NEXT_STEP 최종 반영 (스캔 동기화)
; L209
LOAD      F00099
MOV       D00001 D00000	// 다음스텝 초기0 차기 Step / 자동스텝 초기0 현재 Step

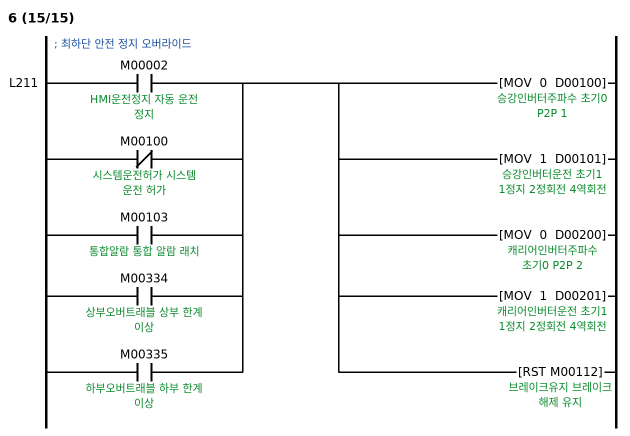
// 최하단 안전 정지 오버라이드
; L211
LOAD      M00002	// HMI운전정지 자동 운전 정지
OR NOT    M00100	// 시스템운전허가 시스템 운전 허가
OR        M00103	// 통합알람 통합 알람 래치
OR        M00334	// 상부오버트래블 상부 한계 이상
OR        M00335	// 하부오버트래블 하부 한계 이상
MOV       0 D00100	// 승강인버터주파수 초기0 P2P 1
MOV       1 D00101	// 승강인버터운전 초기1 1정지 2정회전 4역회전
MOV       0 D00200	// 캐리어인버터주파수 초기0 P2P 2
MOV       1 D00201	// 캐리어인버터운전 초기1 1정지 2정회전 4역회전
RST       M00112	// 브레이크유지 브레이크 해제 유지

VARIABLES AND COMMENTS (devices not used above)
P00027	BIT	브레이크해제 // 승강 브레이크 해제
D00020	WORD	승강고속주파수 // 초기5000 50Hz
P00026	BIT	알람램프부저 // 통합 알람 출력
P00024	BIT	운전램프 // 운전 상태 표시
T0011	BIT/WORD	인입타임아웃 // 설정150 15초
P00025	BIT	정지램프 // 정지 상태 표시
P00020	BIT	층1입고컨베이어 // 1층 입고 컨베이어
P00021	BIT	층2출고컨베이어 // 2층 출고 컨베이어
P00022	BIT	층3출고컨베이어 // 3층 출고 컨베이어
P00023	BIT	층4출고컨베이어 // 4층 출고 컨베이어
T0001	BIT/WORD	화물안착타이머 // 설정5 0.5초